TYPE RobotData :
STRUCT
	//Variables will be manipulated by Unity via ADS
	targetX : INT;
	targetY : INT;
	targetZ : INT;	
	velocity : INT;	//Global value for all joints
	
	joint0 : Joint;
	joint1 : Joint;
	joint2 : Joint;
	joint3 : Joint;
	joint4 : Joint;
	
	
END_STRUCT
END_TYPE

(* stored: Version 1.1.0.1, ProductVersion 3.1.4024.12
   DUT RobotData: Id {ba5a1984-06db-40e2-af22-f49ed11fba5f} *)
